{attribute 'qualified_only'}
VAR_GLOBAL PERSISTENT
	
	astEventsHistory			: ARRAY[0..200] OF ST_EventsHistory;
	
END_VAR

(* stored: Version 1.1.0.1
   GVL GVL_Persistent: Id {c4e2d847-c262-4f9e-8eeb-2ef378462b76} *)
